Yaskawa INFORM job: FRONT_SEARCH_90ST-2_5140.JBI

/JOB
//NAME FRONT_SEARCH_90ST-2_5140
///FOLDERNAME 02-SKRZYNIE_JOBS
//POS
///NPOS 32,32,0,5,0,0
///TOOL 0
///POSTYPE PULSE
///PULSE
C00000=-24267,-14312,28258,73734,-14690,6801
C00001=-48856,-20471,20184,80604,22934,-693
C00002=-64684,-12387,-4503,43203,44892,28767
C00003=-66627,-3447,7116,44802,44939,27584
C00004=-65533,-2317,8306,44379,44431,27933
C00005=-67334,-2160,8474,45030,45313,27386
C00006=-67334,-1447,10904,45827,44533,26848
C00007=-67334,-2160,8474,45030,45313,27386
C00008=-39493,-23395,-11743,31695,31554,37072
C00009=-35655,-22301,-10918,28352,30443,39151
C00010=-36960,-21613,-9866,29618,30701,38377
C00011=-35744,-19595,-8276,28251,30660,39198
C00012=-36810,-20242,-8792,29253,30902,38584
C00013=-36810,-19249,-5623,30469,29669,37920
C00014=-36810,-20242,-8792,29253,30902,38584
C00015=19451,-23723,-4446,126880,-27266,-2952
C00016=19498,-23692,-4078,126522,-27139,-2758
C00017=19135,-22655,-3320,127123,-27127,-3111
C00018=19251,-22842,-3139,126667,-27009,-2858
C00019=19251,-21966,-656,125111,-26336,-2039
C00020=19690,-24221,-4457,126204,-27147,-2571
C00021=19623,-34877,-16768,124729,-29078,51940
C00022=15304,-25293,-919,164625,-9673,28990
C00023=15060,-24487,-364,165662,-9870,28471
C00024=14820,-23667,211,166639,-10065,27982
C00025=14946,-24106,-99,166125,-9960,28239
C00026=14946,-23268,2164,165268,-9043,28646
C00027=15172,-24866,-626,165185,-9778,28711
C00028=22935,-43287,-23487,146875,-13252,38235
C00029=53252,-41973,-2905,102185,-37459,42403
C00030=0,-35574,42087,36666,-9339,1809
C00031=0,-52278,40443,0,6873,1
BC00000=938167
BC00001=938167
BC00002=970052
BC00003=970052
BC00004=970052
BC00005=970052
BC00006=970052
BC00007=970052
BC00008=970052
BC00009=970052
BC00010=970052
BC00011=970052
BC00012=970052
BC00013=970052
BC00014=970052
BC00015=970052
BC00016=970052
BC00017=970052
BC00018=970052
BC00019=970052
BC00020=970052
BC00021=970052
BC00022=970052
BC00023=970052
BC00024=970052
BC00025=970052
BC00026=970052
BC00027=970052
BC00028=956686
BC00029=911348
BC00030=796997
BC00031=790120
///POSTYPE BASE
///RECTAN
///RCONF 1,0,0,0,0,0,0,0,0,0,0,0,0,0,0,0,0,0,0,0,0,0,0,0
P00006=0.000,0.000,0.000,0.0000,0.0000,0.0000
///RCONF 0,0,0,0,0,0,0,0,0,0,0,0,0,0,0,0,0,0,0,0,0,0,0,0
P00501=-2.026,0.009,3.534,0.0000,0.0000,0.0000
///RCONF 1,0,0,0,0,0,0,0,0,0,0,0,0,0,0,0,0,0,0,0,0,0,0,0
P00502=-2.023,0.001,1.732,0.0000,0.0000,0.0000
P00503=0.138,-0.044,1.539,0.0000,0.0000,0.0000
P00504=-0.309,-0.010,1.636,0.0000,0.0000,0.0000
//INST
///DATE 2024/05/26 15:08
///ATTR SC,RW
///GROUP1 RB1,BS1
NOP
MOVJ C00000 BC00000 VJ=80.00
MOVJ C00001 BC00001 VJ=40.00
'::::::::::::::::::::::::::::::::
'W56 P
'::::::::::::::::::::::::::::::::
MOVL C00002 BC00002 V=500.0
SFTOF
MOVL C00003 BC00003 V=166.7 PL=0
REFP 3 C00004 BC00004
CALL JOB:SEARCH-R1
SET P0501 P0006
SFTON P0501
MOVL C00005 BC00005 V=166.7 PL=0
REFP 3 C00006 BC00006
CALL JOB:SEARCH-R1
SET P0501 P0006
SFTON P0501
MOVL C00007 BC00007 V=250.0 PL=0
SFTOF
MOVL C00008 BC00008 V=333.3
'::::::::::::::::::::::::::::::::
'W56 L
'::::::::::::::::::::::::::::::::
MOVL C00009 BC00009 V=333.3
MOVL C00010 BC00010 V=166.7 PL=0
REFP 3 C00011 BC00011
CALL JOB:SEARCH-R1
SET P0502 P0006
SFTON P0502
MOVL C00012 BC00012 V=166.7 PL=0
REFP 3 C00013 BC00013
CALL JOB:SEARCH-R1
SET P0502 P0006
SFTON P0502
MOVL C00014 BC00014 V=250.0 PL=0
SFTOF
'::::::::::::::::::::::::::::::::
'W57 P
'::::::::::::::::::::::::::::::::
MOVL C00015 BC00015 V=500.0
MOVL C00016 BC00016 V=100.0 PL=0
REFP 3 C00017 BC00017
CALL JOB:SEARCH-R1
SET P0503 P0006
SFTON P0503
MOVL C00018 BC00018 V=166.7 PL=0
REFP 3 C00019 BC00019
CALL JOB:SEARCH-R1
SET P0503 P0006
SFTON P0503
MOVL C00020 BC00020 V=250.0 PL=0
SFTOF
'::::::::::::::::::::::::::::::::
'W57 L
'::::::::::::::::::::::::::::::::
MOVL C00021 BC00021 V=333.3
MOVL C00022 BC00022 V=500.0
MOVL C00023 BC00023 V=166.7 PL=0
REFP 3 C00024 BC00024
CALL JOB:SEARCH-R1
SET P0504 P0006
SFTON P0504
MOVL C00025 BC00025 V=166.7 PL=0
REFP 3 C00026 BC00026
CALL JOB:SEARCH-R1
SET P0504 P0006
SFTON P0504
MOVL C00027 BC00027 V=250.0 PL=0
SFTOF
MOVJ C00028 BC00028 VJ=50.00
MOVJ C00029 BC00029 VJ=50.00
MOVJ C00030 BC00030 VJ=80.00
MOVJ C00031 BC00031 VJ=80.00
END
